FUNCTION_BLOCK PusherControllerIProv (* Pusher Controller Interface Provider *)
  (* Standard: 61499-2 *)
  (* Version 0.2, 2003-12-05, JHC, Rockwell Automation, Renamed from NEWCOMPFB. *)
  (* Version 0.1, 2002-01-08, JHC, Rockwell Automation, Added DLY FB as example. *)
  (* Version 0.0, 2000-05-27, JHC, Rockwell Automation *)
  (* Compiler header: package fb.rt.dasdA1.A2.Pusher; *)
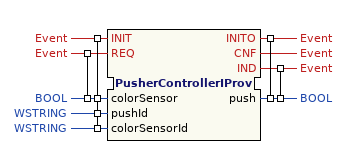
  EVENT_INPUT
    INIT WITH colorSensor, pushId, colorSensorId; (* Initialization Request *)
    REQ WITH colorSensor; (* Normal Execution Request *)
  END_EVENT
  EVENT_OUTPUT
    INITO WITH push; (* Initialization Confirm *)
    CNF; (* Execution Confirmation *)
    IND WITH push;
  END_EVENT
  VAR_INPUT
    colorSensor : BOOL; (* Status of Color sensor *)
    pushId : WSTRING; (* Push event id *)
    colorSensorId : WSTRING; (* Id of the color sensor *)
  END_VAR
  VAR_OUTPUT
    push : BOOL;
  END_VAR
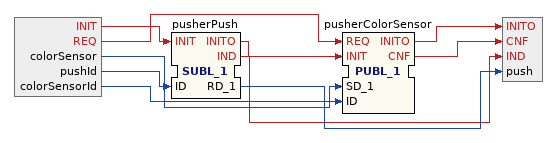
  FBS
    pusherColorSensor : PUBL_1;
    pusherPush : SUBL_1;
  END_FBS
  EVENT_CONNECTIONS
    REQ TO pusherColorSensor.REQ;
    pusherColorSensor.INITO TO INITO;
    pusherPush.INITO TO pusherColorSensor.INIT;
    INIT TO pusherPush.INIT;
    pusherColorSensor.CNF TO CNF;
    pusherPush.IND TO IND;
  END_CONNECTIONS
  DATA_CONNECTIONS
    colorSensor TO pusherColorSensor.SD_1;
    colorSensorId TO pusherColorSensor.ID;
    pushId TO pusherPush.ID;
    pusherPush.RD_1 TO push;
  END_CONNECTIONS
END_FUNCTION_BLOCK
